// {attribute 'hide_all_locals'}
FUNCTION_BLOCK FB_Huawei_SmartLogger
VAR_INPUT PERSISTENT
	bEnable						: BOOL;				//True = Function is enabled, FALSE = Function is dissabled, no new Data
	sIPAdress					: STRING(15);		//IP Adress from the Inverter
	sint_ID_Iverter1			:SINT;				// ID of inveter 1
	sint_ID_Iverter2			:SINT;				// ID of inveter 2
	sint_ID_Iverter3			:SINT;				// ID of inveter 3
	sint_ID_Iverter4			:SINT;				// ID of inveter 4
	sint_ID_Iverter5			:SINT;				// ID of inveter 5
	sint_ID_Iverter6			:SINT;				// ID of inveter 6
	sint_ID_Iverter7			:SINT;				// ID of inveter 7
	sint_ID_Iverter8			:SINT;				// ID of inveter 8
	sint_ID_Iverter9			:SINT;				// ID of inveter 9
	sint_ID_Iverter10			:SINT;				// ID of inveter 10
	sint_ID_Iverter11			:SINT;				// ID of inveter 11
	sint_ID_Iverter12			:SINT;				// ID of inveter 12
	
	
END_VAR
VAR_OUTPUT
	st_Huawei_SmartLogger		: ARRAY[1..20] OF ST_Huawei_SmartLogger_OutData;					//Output structure with Data 
	stDataEMPower_PV			: ARRAY[1..20] OF ST_ElectricMeter_Output_Power;					//Output structure with Data from Electric Meter PV (Power Data)
	stDataEMCounter_PV 			: ARRAY[1..20] OF ST_ElectricMeter_Output_Counter;					//Output structure with Data from Electric Meter PV (Counter Data)
	diNrOfEM_OUT_PV				: DINT;																//Active Number from the Electric Meter for using on other functions
END_VAR
VAR
	sint_ID_Iverter				:ARRAY[1..12] OF SINT;				// Array of ID of inveter 
	fbMeter						: ARRAY[1..30] OF FB_ElectricMeter;					//Electric Meter Function 
	fbElMeter					: FB_ElectricMeter;									//Electric Meter Function for sumation values 
	
	fbNumberDevice				: FB_NumberOfDevice;								//Function block to calcualte the number of the Device
	fbConvertEnergyRegister		: FB_CV_WORD_TO_DWORD;								//Convert function
	fbMBRead_FC3				: FB_MBReadRegs;									//Modbus Read Function (FC3)
	timDelay					: TON;												//Timer for Delay between Requests
	timTimeout					: TON;												//Timer for Timeout
	timDissableFunctions		: TON;												//Timer to dissable the Function after Lynus_Standards.Constants_General.tTimeDissableLynusFunctions Days without connection to the Lynus Cloud
	timResetConnectionOnGVL		: TON;												//Timer to try reset the connection Flag on the GVL. (When somebody delete the Connection Function and make only a onlinechange)
	FPEnable					: R_TRIG;											//Internal positive Edge
	FPError_FC_3				: R_TRIG;											//Internal positive Edge
	PD_String					: FB_PersistentData_String;							//Function to save persistent data 
	stFloat						: ST_UN_FLOAT_CONVERT_DWORD_REAL;					//Convert the Float Raw Value
	arrBuffer_FC3				: ARRAY[0..25] OF WORD;							//Buffer with Data from FC3
	arrPD						: ARRAY[1..2] OF FB_PersistentData_Number;			//Function to save persistent data 
	byWaitInStep				: BYTE;												//Wait in Step before start to clean data on PLC
	iStateGVLData				: INT;												//State machine to handle the data on the GVL
	iStateModbus				: INT;												//State variable for Statemachine
	iStateModbus_CP				: INT;												//Compare State variable
	diCounterForGVL				: DINT;												//Counter to clean old data on GVL
	lrCheckValue				: LREAL;											//Internal Value to check the value before convert
	x							: INT;
	i: INT;
	int_Poll_Counter			: INT;												//Poll1 = inverter_ID 1,....
	byLPForInverter: INT;
	lrCounterEnergyProduction: LREAL;
	dwInput: DWORD;
	int_maxPolls				:INT :=12;											//maximum number of polls / inverter. 
	ton_Wait: Ton;
	FB_ConvertData			:FB_Convert_Huawei_SmartLogger;
	lreal1: LREAL;
	lreal2: LREAL;
	lreal3: LREAL;
	lreal4: LREAL;
	lreal5: LREAL;
	lreal6: LREAL;
	lreal7: LREAL;
	lreal8: LREAL;
	lreal9: LREAL;
	lreal10: LREAL;
	lreal11: LREAL;
	lreal12: LREAL;
	lreal13: LREAL;
	lreal14: LREAL;
	lreal15: LREAL;
	lreal16: LREAL;
	lreal17: LREAL;
	lreal18: LREAL;
	lreal19: LREAL;
	lreal20: LREAL;
	END_VAR

//Creator : Stefan Lackner
//Company : EfficientIO
//Date : 17.10.2022
//Version : 0.0.0.1		

//With this function its possible to read out values from the SmartLogger from the manufacturer Huawei
//This Function read out the Values from up to 12 inverters behind a SmartLogger. The SmartLogger could handle up to 247 inverters. 
//The protocol to the Inverter is Modbus TCP
//Attention. To access the registers, an offset of 1 must always be subtracted. Register 40001 would then be on register 40000.
//The document "SmartLogger ModBus Interface Definitions.pdf" issue 35 got used for the Modbus adress List

//NOTE for diNr.....Designation => 
//_IN = Here Data come in from other Functions or go out to other functions about the GVL
//_OUT = Here Data go out to other functions about the GVL


(*------------------------------------------------------------------------------------------General Input Part---------------------------------------------------------------------------------------------*)

//Check limitation
sint_ID_Iverter1 := LIMIT(0,sint_ID_Iverter1,127);
sint_ID_Iverter2 := LIMIT(0,sint_ID_Iverter2,127);
sint_ID_Iverter3 := LIMIT(0,sint_ID_Iverter3,127);
sint_ID_Iverter4 := LIMIT(0,sint_ID_Iverter4,127);
sint_ID_Iverter5 := LIMIT(0,sint_ID_Iverter5,127);
sint_ID_Iverter6 := LIMIT(0,sint_ID_Iverter6,127);
sint_ID_Iverter7 := LIMIT(0,sint_ID_Iverter7,127);
sint_ID_Iverter8 := LIMIT(0,sint_ID_Iverter8,127);
sint_ID_Iverter9 := LIMIT(0,sint_ID_Iverter9,127);
sint_ID_Iverter10:= LIMIT(0,sint_ID_Iverter10,127);
sint_ID_Iverter11:= LIMIT(0,sint_ID_Iverter11,127);
sint_ID_Iverter12 := LIMIT(0,sint_ID_Iverter12,127);
// copy in an array, easier for handling in the state maschine
sint_ID_Iverter[1]	:=	sint_ID_Iverter1;
sint_ID_Iverter[2]	:=	sint_ID_Iverter2;
sint_ID_Iverter[3]	:=	sint_ID_Iverter3;
sint_ID_Iverter[4]	:=	sint_ID_Iverter4;
sint_ID_Iverter[5]	:=	sint_ID_Iverter5;
sint_ID_Iverter[6]	:=	sint_ID_Iverter6;
sint_ID_Iverter[7]	:=	sint_ID_Iverter7;
sint_ID_Iverter[8]	:=	sint_ID_Iverter8;
sint_ID_Iverter[9]	:=	sint_ID_Iverter9;
sint_ID_Iverter[10]	:=	sint_ID_Iverter10;
sint_ID_Iverter[11]	:=	sint_ID_Iverter11;
sint_ID_Iverter[12]	:=	sint_ID_Iverter12;



(*-------------------------------------------------------------Calcualte the number of EM System---------------------------------------------------------------*)

fbNumberDevice(
	diActualNumberOfDevices:= Lynus_Standards.GVL_Energy.stNumberOfDevices.diNumberOfElectricMeters, 
	diMaxNumberOfDevices:= Constants_Energy.diMaxNumberOfElectricMeters, 
	udiCounterOnlineChange:= TwinCAT_SystemInfoVarList._AppInfo.OnlineChangeCnt, 
	bNumberIsCalculatet=> , 
	bFPNumberIsCalculatet=> , 
	bOnlineChange=> , 
	diNumberForThisDevice=> diNrOfEM_OUT_PV, 
	diNumberOfTotalDevices=> );

//Write new Numer on GVL
IF fbNumberDevice.bFPNumberIsCalculatet THEN
	Lynus_Standards.GVL_Energy.stNumberOfDevices.diNumberOfElectricMeters := fbNumberDevice.diNumberOfTotalDevices;	
END_IF 

//Delete old Number on GVL
IF fbNumberDevice.bOnlineChange THEN 
	Lynus_Standards.GVL_Energy.stNumberOfDevices.diNumberOfElectricMeters := diNrOfEM_OUT_PV;	
		iStateGVLData := 1; 
END_IF

(*-------------------------------------------------------------Service from Backend is ready and check the connection to backend for dissabel/enable Function---------------------------------------------------------------*)

//Try to reset the variable for connection on the GVL. When all is normal then the EfficientIO Mqtt connection function set this variable to true in the next cycle
//When we have no connection to the backend then after Lynus_Standards.Constants_General.tTimeDissableLynusFunctions days the Function is dissabled with all of his functionalities
timResetConnectionOnGVL(IN:= NOT timResetConnectionOnGVL.Q, PT:= T#1H, Q=> , ET=> );
IF timResetConnectionOnGVL.Q THEN 
	Lynus_Standards.GVL_Communicator.bStateConnectionToEnableFunctions := FALSE; 
END_IF
IF NOT Lynus_Standards.GVL_Communicator.bStateConnectionToEnableFunctions THEN 
	timDissableFunctions.IN := TRUE; 
ELSE 
	timDissableFunctions.IN := FALSE; 
END_IF  
timDissableFunctions(IN:= , PT:= Lynus_Standards.Constants_General.tTimeDissableLynusFunctions, Q=> , ET=> );
	
(*------------------------------------------------------------------------------------------State Machine---------------------------------------------------------------------------------------------*)
	
//Enable
FPEnable(CLK:= bEnable, Q=> );
IF FPEnable.Q AND iStateModbus = 0 THEN 
	iStateModbus := 1; 
END_IF
IF NOT bEnable OR timDissableFunctions.Q THEN 
	iStateModbus := 0; 
END_IF

//Timer for delay
timDelay(IN:= , PT:= T#100MS, Q=> , ET=> );	

//Timer for Timeout in Statemachine
IF iStateModbus = iStateModbus_CP THEN 
	timTimeout.IN := TRUE; 
ELSE 
	timTimeout.IN := FALSE; 
END_IF
IF iStateModbus = 0 THEN 
	timTimeout.IN := FALSE; 
END_IF
timTimeout(IN:= , PT:= T#20S, Q=> , ET=> );	


//Statemachine
CASE iStateModbus OF
	
	0://Init Step
		iStateModbus_CP := iStateModbus;
		timDelay.IN := FALSE;
		FOR i:=1 TO 20 BY 1 DO
			st_Huawei_SmartLogger[i].bFunctionIsActive := FALSE;
			st_Huawei_SmartLogger[i].eOperatingStateInverter := E_Huawei_SmartLogger_OperatingState.Unknown ;
		END_FOR
		
		fbMBRead_FC3.bExecute := FALSE;
		lrCheckValue := 0;
									
	1://Read out first inverter
		int_Poll_Counter:=1;			//Poll int_Poll_Counter : Inverter int_Poll_Counter 	
		st_Huawei_SmartLogger[int_Poll_Counter].bFunctionIsActive := TRUE;
		iStateModbus_CP := iStateModbus;
		fbMBRead_FC3.nQuantity := 25;
		fbMBRead_FC3.nMBAddr := (51000+(25*(SINT_TO_WORD(sint_ID_Iverter[int_Poll_Counter]) - 1)));
		fbMBRead_FC3.bExecute := TRUE;
			
		IF fbMBRead_FC3.bBusy THEN 
			timDelay.IN := TRUE; 
		END_IF
		
		//Wait for Delay, copy Data and then next step
		IF NOT fbMBRead_FC3.bBusy AND NOT fbMBRead_FC3.bError AND timDelay.Q THEN
			// convert received data
			FB_ConvertData(	arrBuffer_FC3			:=	arrBuffer_FC3,
											int_Poll_Counter		:=	int_Poll_Counter,
											lrPowerTotal			=>	fbMeter[int_Poll_Counter].lrPowerTotal,	
											lrReactivePowerTotal	=> 	fbMeter[int_Poll_Counter].lrReactivePowerTotal,
											eOperatingStateInverter	=>	st_Huawei_SmartLogger[int_Poll_Counter].eOperatingStateInverter);
	
			//Next Step
			fbMBRead_FC3.bExecute := FALSE;
			timDelay.IN := FALSE;
			iStateModbus := iStateModbus+1;
			IF arrBuffer_FC3[9]<>0 THEN
				st_Huawei_SmartLogger[int_Poll_Counter].bError := FALSE; 
				st_Huawei_SmartLogger[int_Poll_Counter].eErrorState := E_Huawei_SmartLogger_Error.eNoError;
			ELSE
				st_Huawei_SmartLogger[int_Poll_Counter].bError := FALSE; 
				st_Huawei_SmartLogger[int_Poll_Counter].eErrorState := E_Huawei_SmartLogger_Error.eNoError;
			END_IF
		END_IF
			
		//Error from Inverter 
		IF NOT fbMBRead_FC3.bBusy AND NOT fbMBRead_FC3.bError AND timDelay.Q AND arrBuffer_FC3[9] >= 16#0300 AND arrBuffer_FC3[9] <= 16#0308 THEN
			iStateModbus := 300;
			st_Huawei_SmartLogger[int_Poll_Counter].eErrorState := E_Huawei_SmartLogger_Error.eHuawei_SmartLoggerError;
		END_IF
	
		//Error or Timeout
		IF FPError_FC_3.Q OR timTimeout.Q THEN
			iStateModbus := 300;
			st_Huawei_SmartLogger[int_Poll_Counter].eOperatingStateInverter := E_Huawei_SmartLogger_OperatingState.Unknown;
			st_Huawei_SmartLogger[int_Poll_Counter].eErrorState	:=	E_Huawei_SmartLogger_Error.eModbusTCPError;
		END_IF
		
	2://Wait and go to step 1 or step 3
		iStateModbus_CP := iStateModbus;
		IF sint_ID_Iverter[int_Poll_Counter+1] = 0 OR int_Poll_Counter=int_maxPolls THEN		// if ID is not in use, go to state 100
			iStateModbus := 100;
		ELSE
			iStateModbus := 3;
			int_Poll_Counter:=int_Poll_Counter+1;			//Poll int_Poll_Counter : Inverter int_Poll_Counter 	
		END_IF

	3://Read out next inverter
		st_Huawei_SmartLogger[int_Poll_Counter].bFunctionIsActive := TRUE;
		iStateModbus_CP := iStateModbus;
		fbMBRead_FC3.nQuantity := 25;
		fbMBRead_FC3.nMBAddr := (51000+(25*(SINT_TO_WORD(sint_ID_Iverter[int_Poll_Counter]) - 1)));
		fbMBRead_FC3.bExecute := TRUE;
			
		IF fbMBRead_FC3.bBusy THEN 
			timDelay.IN := TRUE; 
		END_IF
		
		//Wait for Delay, copy Data and then next step
		IF NOT fbMBRead_FC3.bBusy AND NOT fbMBRead_FC3.bError AND timDelay.Q THEN
			// convert received data
			FB_ConvertData(	arrBuffer_FC3			:=	arrBuffer_FC3,
											int_Poll_Counter		:=	int_Poll_Counter,
											lrPowerTotal			=>	fbMeter[int_Poll_Counter].lrPowerTotal,	
											lrReactivePowerTotal	=> 	fbMeter[int_Poll_Counter].lrReactivePowerTotal,
											eOperatingStateInverter	=>	st_Huawei_SmartLogger[int_Poll_Counter].eOperatingStateInverter);
	
			//Next Step
			fbMBRead_FC3.bExecute := FALSE;
			timDelay.IN := FALSE;
			iStateModbus := iStateModbus+1;
			IF arrBuffer_FC3[9]<>0 THEN
				st_Huawei_SmartLogger[int_Poll_Counter].bError := FALSE; 
				st_Huawei_SmartLogger[int_Poll_Counter].eErrorState := E_Huawei_SmartLogger_Error.eNoError;
			ELSE
				st_Huawei_SmartLogger[int_Poll_Counter].bError := FALSE; 
				st_Huawei_SmartLogger[int_Poll_Counter].eErrorState := E_Huawei_SmartLogger_Error.eNoError;
			END_IF
		END_IF
			
		//Error from Inverter 
		IF NOT fbMBRead_FC3.bBusy AND NOT fbMBRead_FC3.bError AND timDelay.Q AND arrBuffer_FC3[9] >= 16#0300 AND arrBuffer_FC3[9] <= 16#0308 THEN
			iStateModbus := 300;
			st_Huawei_SmartLogger[int_Poll_Counter].eErrorState := E_Huawei_SmartLogger_Error.eHuawei_SmartLoggerError;
		END_IF
	
		//Error or Timeout
		IF FPError_FC_3.Q OR timTimeout.Q THEN
			iStateModbus := 300;
			st_Huawei_SmartLogger[int_Poll_Counter].eOperatingStateInverter := E_Huawei_SmartLogger_OperatingState.Unknown;
			st_Huawei_SmartLogger[int_Poll_Counter].eErrorState	:=	E_Huawei_SmartLogger_Error.eModbusTCPError;
		END_IF
		
	4://Wait and go to step +1 or step 100
		iStateModbus_CP := iStateModbus;
		IF sint_ID_Iverter[int_Poll_Counter+1] = 0 OR int_Poll_Counter=int_maxPolls THEN		// if ID is not in use, go to state 100
			iStateModbus := 100;
		ELSE
			iStateModbus := iStateModbus+1;
			int_Poll_Counter:=int_Poll_Counter+1;			//Poll int_Poll_Counter : Inverter int_Poll_Counter 	
		END_IF
	
	5://Read out next inverter
		st_Huawei_SmartLogger[int_Poll_Counter].bFunctionIsActive := TRUE;
		iStateModbus_CP := iStateModbus;
		fbMBRead_FC3.nQuantity := 25;
		fbMBRead_FC3.nMBAddr := (51000+(25*(SINT_TO_WORD(sint_ID_Iverter[int_Poll_Counter]) - 1)));
		fbMBRead_FC3.bExecute := TRUE;
			
		IF fbMBRead_FC3.bBusy THEN 
			timDelay.IN := TRUE; 
		END_IF
		
		//Wait for Delay, copy Data and then next step
		IF NOT fbMBRead_FC3.bBusy AND NOT fbMBRead_FC3.bError AND timDelay.Q THEN
			// convert received data
			FB_ConvertData(	arrBuffer_FC3			:=	arrBuffer_FC3,
											int_Poll_Counter		:=	int_Poll_Counter,
											lrPowerTotal			=>	fbMeter[int_Poll_Counter].lrPowerTotal,	
											lrReactivePowerTotal	=> 	fbMeter[int_Poll_Counter].lrReactivePowerTotal,
											eOperatingStateInverter	=>	st_Huawei_SmartLogger[int_Poll_Counter].eOperatingStateInverter);
	
			//Next Step
			fbMBRead_FC3.bExecute := FALSE;
			timDelay.IN := FALSE;
			iStateModbus := iStateModbus+1;
			IF arrBuffer_FC3[9]<>0 THEN
				st_Huawei_SmartLogger[int_Poll_Counter].bError := FALSE; 
				st_Huawei_SmartLogger[int_Poll_Counter].eErrorState := E_Huawei_SmartLogger_Error.eNoError;
			ELSE
				st_Huawei_SmartLogger[int_Poll_Counter].bError := FALSE; 
				st_Huawei_SmartLogger[int_Poll_Counter].eErrorState := E_Huawei_SmartLogger_Error.eNoError;
			END_IF
		END_IF
			
		//Error from Inverter 
		IF NOT fbMBRead_FC3.bBusy AND NOT fbMBRead_FC3.bError AND timDelay.Q AND arrBuffer_FC3[9] >= 16#0300 AND arrBuffer_FC3[9] <= 16#0308 THEN
			iStateModbus := 300;
			st_Huawei_SmartLogger[int_Poll_Counter].eErrorState := E_Huawei_SmartLogger_Error.eHuawei_SmartLoggerError;
		END_IF
	
		//Error or Timeout
		IF FPError_FC_3.Q OR timTimeout.Q THEN
			iStateModbus := 300;
			st_Huawei_SmartLogger[int_Poll_Counter].eOperatingStateInverter := E_Huawei_SmartLogger_OperatingState.Unknown;
			st_Huawei_SmartLogger[int_Poll_Counter].eErrorState	:=	E_Huawei_SmartLogger_Error.eModbusTCPError;
		END_IF
		
	6://Wait and go to step +1 or step 100
		iStateModbus_CP := iStateModbus;
		IF sint_ID_Iverter[int_Poll_Counter+1] = 0 OR int_Poll_Counter=int_maxPolls THEN		// if ID is not in use, go to state 100
			iStateModbus := 100;
		ELSE
			iStateModbus := iStateModbus+1;
			int_Poll_Counter:=int_Poll_Counter+1;			//Poll int_Poll_Counter : Inverter int_Poll_Counter 	
		END_IF
		
	7://Read out next inverter
		st_Huawei_SmartLogger[int_Poll_Counter].bFunctionIsActive := TRUE;
		iStateModbus_CP := iStateModbus;
		fbMBRead_FC3.nQuantity := 25;
		fbMBRead_FC3.nMBAddr := (51000+(25*(SINT_TO_WORD(sint_ID_Iverter[int_Poll_Counter]) - 1)));
		fbMBRead_FC3.bExecute := TRUE;
			
		IF fbMBRead_FC3.bBusy THEN 
			timDelay.IN := TRUE; 
		END_IF
		
		//Wait for Delay, copy Data and then next step
		IF NOT fbMBRead_FC3.bBusy AND NOT fbMBRead_FC3.bError AND timDelay.Q THEN
			// convert received data
			FB_ConvertData(	arrBuffer_FC3			:=	arrBuffer_FC3,
											int_Poll_Counter		:=	int_Poll_Counter,
											lrPowerTotal			=>	fbMeter[int_Poll_Counter].lrPowerTotal,	
											lrReactivePowerTotal	=> 	fbMeter[int_Poll_Counter].lrReactivePowerTotal,
											eOperatingStateInverter	=>	st_Huawei_SmartLogger[int_Poll_Counter].eOperatingStateInverter);
	
			//Next Step
			fbMBRead_FC3.bExecute := FALSE;
			timDelay.IN := FALSE;
			iStateModbus := iStateModbus+1;
			IF arrBuffer_FC3[9]<>0 THEN
				st_Huawei_SmartLogger[int_Poll_Counter].bError := FALSE; 
				st_Huawei_SmartLogger[int_Poll_Counter].eErrorState := E_Huawei_SmartLogger_Error.eNoError;
			ELSE
				st_Huawei_SmartLogger[int_Poll_Counter].bError := FALSE; 
				st_Huawei_SmartLogger[int_Poll_Counter].eErrorState := E_Huawei_SmartLogger_Error.eNoError;
			END_IF
		END_IF
			
		//Error from Inverter 
		IF NOT fbMBRead_FC3.bBusy AND NOT fbMBRead_FC3.bError AND timDelay.Q AND arrBuffer_FC3[9] >= 16#0300 AND arrBuffer_FC3[9] <= 16#0308 THEN
			iStateModbus := 300;
			st_Huawei_SmartLogger[int_Poll_Counter].eErrorState := E_Huawei_SmartLogger_Error.eHuawei_SmartLoggerError;
		END_IF
	
		//Error or Timeout
		IF FPError_FC_3.Q OR timTimeout.Q THEN
			iStateModbus := 300;
			st_Huawei_SmartLogger[int_Poll_Counter].eOperatingStateInverter := E_Huawei_SmartLogger_OperatingState.Unknown;
			st_Huawei_SmartLogger[int_Poll_Counter].eErrorState	:=	E_Huawei_SmartLogger_Error.eModbusTCPError;
		END_IF

	8://Wait and go to step +1 or step 100
		iStateModbus_CP := iStateModbus;
		IF sint_ID_Iverter[int_Poll_Counter+1] = 0 OR int_Poll_Counter=int_maxPolls THEN		// if ID is not in use, go to state 100
			iStateModbus := 100;
		ELSE
			iStateModbus := iStateModbus+1;
			int_Poll_Counter:=int_Poll_Counter+1;			//Poll int_Poll_Counter : Inverter int_Poll_Counter 	
		END_IF
		
	9://Read out next inverter
		st_Huawei_SmartLogger[int_Poll_Counter].bFunctionIsActive := TRUE;
		iStateModbus_CP := iStateModbus;
		fbMBRead_FC3.nQuantity := 25;
		fbMBRead_FC3.nMBAddr := (51000+(25*(SINT_TO_WORD(sint_ID_Iverter[int_Poll_Counter]) - 1)));
		fbMBRead_FC3.bExecute := TRUE;
			
		IF fbMBRead_FC3.bBusy THEN 
			timDelay.IN := TRUE; 
		END_IF
		
		//Wait for Delay, copy Data and then next step
		IF NOT fbMBRead_FC3.bBusy AND NOT fbMBRead_FC3.bError AND timDelay.Q THEN
			// convert received data
			FB_ConvertData(	arrBuffer_FC3			:=	arrBuffer_FC3,
											int_Poll_Counter		:=	int_Poll_Counter,
											lrPowerTotal			=>	fbMeter[int_Poll_Counter].lrPowerTotal,	
											lrReactivePowerTotal	=> 	fbMeter[int_Poll_Counter].lrReactivePowerTotal,
											eOperatingStateInverter	=>	st_Huawei_SmartLogger[int_Poll_Counter].eOperatingStateInverter);
	
			//Next Step
			fbMBRead_FC3.bExecute := FALSE;
			timDelay.IN := FALSE;
			iStateModbus := iStateModbus+1;
			IF arrBuffer_FC3[9]<>0 THEN
				st_Huawei_SmartLogger[int_Poll_Counter].bError := FALSE; 
				st_Huawei_SmartLogger[int_Poll_Counter].eErrorState := E_Huawei_SmartLogger_Error.eNoError;
			ELSE
				st_Huawei_SmartLogger[int_Poll_Counter].bError := FALSE; 
				st_Huawei_SmartLogger[int_Poll_Counter].eErrorState := E_Huawei_SmartLogger_Error.eNoError;
			END_IF
		END_IF
			
		//Error from Inverter 
		IF NOT fbMBRead_FC3.bBusy AND NOT fbMBRead_FC3.bError AND timDelay.Q AND arrBuffer_FC3[9] >= 16#0300 AND arrBuffer_FC3[9] <= 16#0308 THEN
			iStateModbus := 300;
			st_Huawei_SmartLogger[int_Poll_Counter].eErrorState := E_Huawei_SmartLogger_Error.eHuawei_SmartLoggerError;
		END_IF
	
		//Error or Timeout
		IF FPError_FC_3.Q OR timTimeout.Q THEN
			iStateModbus := 300;
			st_Huawei_SmartLogger[int_Poll_Counter].eOperatingStateInverter := E_Huawei_SmartLogger_OperatingState.Unknown;
			st_Huawei_SmartLogger[int_Poll_Counter].eErrorState	:=	E_Huawei_SmartLogger_Error.eModbusTCPError;
		END_IF
		
	10://Wait and go to step +1 or step 100
		iStateModbus_CP := iStateModbus;
		IF sint_ID_Iverter[int_Poll_Counter+1] = 0 OR int_Poll_Counter=int_maxPolls THEN		// if ID is not in use, go to state 100
			iStateModbus := 100;
		ELSE
			iStateModbus := iStateModbus+1;
			int_Poll_Counter:=int_Poll_Counter+1;			//Poll int_Poll_Counter : Inverter int_Poll_Counter 	
		END_IF
		
	11://Read out next inverter
		st_Huawei_SmartLogger[int_Poll_Counter].bFunctionIsActive := TRUE;
		iStateModbus_CP := iStateModbus;
		fbMBRead_FC3.nQuantity := 25;
		fbMBRead_FC3.nMBAddr := (51000+(25*(SINT_TO_WORD(sint_ID_Iverter[int_Poll_Counter]) - 1)));
		fbMBRead_FC3.bExecute := TRUE;
			
		IF fbMBRead_FC3.bBusy THEN 
			timDelay.IN := TRUE; 
		END_IF
		
		//Wait for Delay, copy Data and then next step
		IF NOT fbMBRead_FC3.bBusy AND NOT fbMBRead_FC3.bError AND timDelay.Q THEN
			// convert received data
			FB_ConvertData(	arrBuffer_FC3			:=	arrBuffer_FC3,
											int_Poll_Counter		:=	int_Poll_Counter,
											lrPowerTotal			=>	fbMeter[int_Poll_Counter].lrPowerTotal,	
											lrReactivePowerTotal	=> 	fbMeter[int_Poll_Counter].lrReactivePowerTotal,
											eOperatingStateInverter	=>	st_Huawei_SmartLogger[int_Poll_Counter].eOperatingStateInverter);
	
			//Next Step
			fbMBRead_FC3.bExecute := FALSE;
			timDelay.IN := FALSE;
			iStateModbus := iStateModbus+1;
			IF arrBuffer_FC3[9]<>0 THEN
				st_Huawei_SmartLogger[int_Poll_Counter].bError := FALSE; 
				st_Huawei_SmartLogger[int_Poll_Counter].eErrorState := E_Huawei_SmartLogger_Error.eNoError;
			ELSE
				st_Huawei_SmartLogger[int_Poll_Counter].bError := FALSE; 
				st_Huawei_SmartLogger[int_Poll_Counter].eErrorState := E_Huawei_SmartLogger_Error.eNoError;
			END_IF
		END_IF
			
		//Error from Inverter 
		IF NOT fbMBRead_FC3.bBusy AND NOT fbMBRead_FC3.bError AND timDelay.Q AND arrBuffer_FC3[9] >= 16#0300 AND arrBuffer_FC3[9] <= 16#0308 THEN
			iStateModbus := 300;
			st_Huawei_SmartLogger[int_Poll_Counter].eErrorState := E_Huawei_SmartLogger_Error.eHuawei_SmartLoggerError;
		END_IF
	
		//Error or Timeout
		IF FPError_FC_3.Q OR timTimeout.Q THEN
			iStateModbus := 300;
			st_Huawei_SmartLogger[int_Poll_Counter].eOperatingStateInverter := E_Huawei_SmartLogger_OperatingState.Unknown;
			st_Huawei_SmartLogger[int_Poll_Counter].eErrorState	:=	E_Huawei_SmartLogger_Error.eModbusTCPError;
		END_IF
		
	12://Wait and go to step +1 or step 100
		iStateModbus_CP := iStateModbus;
		IF sint_ID_Iverter[int_Poll_Counter+1] = 0 OR int_Poll_Counter=int_maxPolls THEN		// if ID is not in use, go to state 100
			iStateModbus := 100;
		ELSE
			iStateModbus := iStateModbus+1;
			int_Poll_Counter:=int_Poll_Counter+1;			//Poll int_Poll_Counter : Inverter int_Poll_Counter 	
		END_IF
		
	13://Read out next inverter
		st_Huawei_SmartLogger[int_Poll_Counter].bFunctionIsActive := TRUE;
		iStateModbus_CP := iStateModbus;
		fbMBRead_FC3.nQuantity := 25;
		fbMBRead_FC3.nMBAddr := (51000+(25*(SINT_TO_WORD(sint_ID_Iverter[int_Poll_Counter]) - 1)));
		fbMBRead_FC3.bExecute := TRUE;
			
		IF fbMBRead_FC3.bBusy THEN 
			timDelay.IN := TRUE; 
		END_IF
		
		//Wait for Delay, copy Data and then next step
		IF NOT fbMBRead_FC3.bBusy AND NOT fbMBRead_FC3.bError AND timDelay.Q THEN
			// convert received data
			FB_ConvertData(	arrBuffer_FC3			:=	arrBuffer_FC3,
											int_Poll_Counter		:=	int_Poll_Counter,
											lrPowerTotal			=>	fbMeter[int_Poll_Counter].lrPowerTotal,	
											lrReactivePowerTotal	=> 	fbMeter[int_Poll_Counter].lrReactivePowerTotal,
											eOperatingStateInverter	=>	st_Huawei_SmartLogger[int_Poll_Counter].eOperatingStateInverter);
	
			//Next Step
			fbMBRead_FC3.bExecute := FALSE;
			timDelay.IN := FALSE;
			iStateModbus := iStateModbus+1;
			IF arrBuffer_FC3[9]<>0 THEN
				st_Huawei_SmartLogger[int_Poll_Counter].bError := FALSE; 
				st_Huawei_SmartLogger[int_Poll_Counter].eErrorState := E_Huawei_SmartLogger_Error.eNoError;
			ELSE
				st_Huawei_SmartLogger[int_Poll_Counter].bError := FALSE; 
				st_Huawei_SmartLogger[int_Poll_Counter].eErrorState := E_Huawei_SmartLogger_Error.eNoError;
			END_IF
		END_IF
			
		//Error from Inverter 1
		IF NOT fbMBRead_FC3.bBusy AND NOT fbMBRead_FC3.bError AND timDelay.Q AND arrBuffer_FC3[9] >= 16#0300 AND arrBuffer_FC3[9] <= 16#0308 THEN
			iStateModbus := 300;
			st_Huawei_SmartLogger[int_Poll_Counter].eErrorState := E_Huawei_SmartLogger_Error.eHuawei_SmartLoggerError;
		END_IF
	
		//Error or Timeout
		IF FPError_FC_3.Q OR timTimeout.Q THEN
			iStateModbus := 300;
			st_Huawei_SmartLogger[int_Poll_Counter].eOperatingStateInverter := E_Huawei_SmartLogger_OperatingState.Unknown;
			st_Huawei_SmartLogger[int_Poll_Counter].eErrorState	:=	E_Huawei_SmartLogger_Error.eModbusTCPError;
		END_IF
		
	14://Wait and go to step +1 or step 100
		iStateModbus_CP := iStateModbus;
		IF sint_ID_Iverter[int_Poll_Counter+1] = 0 OR int_Poll_Counter=int_maxPolls THEN		// if ID is not in use, go to state 100
			iStateModbus := 100;
		ELSE
			iStateModbus := iStateModbus+1;
			int_Poll_Counter:=int_Poll_Counter+1;			//Poll int_Poll_Counter : Inverter int_Poll_Counter 	
		END_IF
		
	15://Read out next inverter
		st_Huawei_SmartLogger[int_Poll_Counter].bFunctionIsActive := TRUE;
		iStateModbus_CP := iStateModbus;
		fbMBRead_FC3.nQuantity := 25;
		fbMBRead_FC3.nMBAddr := (51000+(25*(SINT_TO_WORD(sint_ID_Iverter[int_Poll_Counter]) - 1)));
		fbMBRead_FC3.bExecute := TRUE;
			
		IF fbMBRead_FC3.bBusy THEN 
			timDelay.IN := TRUE; 
		END_IF
		
		//Wait for Delay, copy Data and then next step
		IF NOT fbMBRead_FC3.bBusy AND NOT fbMBRead_FC3.bError AND timDelay.Q THEN
			// convert received data
			FB_ConvertData(	arrBuffer_FC3			:=	arrBuffer_FC3,
											int_Poll_Counter		:=	int_Poll_Counter,
											lrPowerTotal			=>	fbMeter[int_Poll_Counter].lrPowerTotal,	
											lrReactivePowerTotal	=> 	fbMeter[int_Poll_Counter].lrReactivePowerTotal,
											eOperatingStateInverter	=>	st_Huawei_SmartLogger[int_Poll_Counter].eOperatingStateInverter);
	
			//Next Step
			fbMBRead_FC3.bExecute := FALSE;
			timDelay.IN := FALSE;
			iStateModbus := iStateModbus+1;
			IF arrBuffer_FC3[9]<>0 THEN
				st_Huawei_SmartLogger[int_Poll_Counter].bError := FALSE; 
				st_Huawei_SmartLogger[int_Poll_Counter].eErrorState := E_Huawei_SmartLogger_Error.eNoError;
			ELSE
				st_Huawei_SmartLogger[int_Poll_Counter].bError := FALSE; 
				st_Huawei_SmartLogger[int_Poll_Counter].eErrorState := E_Huawei_SmartLogger_Error.eNoError;
			END_IF
		END_IF
			
		//Error from Inverter 
		IF NOT fbMBRead_FC3.bBusy AND NOT fbMBRead_FC3.bError AND timDelay.Q AND arrBuffer_FC3[9] >= 16#0300 AND arrBuffer_FC3[9] <= 16#0308 THEN
			iStateModbus := 300;
			st_Huawei_SmartLogger[int_Poll_Counter].eErrorState := E_Huawei_SmartLogger_Error.eHuawei_SmartLoggerError;
		END_IF
	
		//Error or Timeout
		IF FPError_FC_3.Q OR timTimeout.Q THEN
			iStateModbus := 300;
			st_Huawei_SmartLogger[int_Poll_Counter].eOperatingStateInverter := E_Huawei_SmartLogger_OperatingState.Unknown;
			st_Huawei_SmartLogger[int_Poll_Counter].eErrorState	:=	E_Huawei_SmartLogger_Error.eModbusTCPError;
		END_IF
		
	16://Wait and go to step +1 or step 100
		iStateModbus_CP := iStateModbus;
		IF sint_ID_Iverter[int_Poll_Counter+1] = 0 OR int_Poll_Counter=int_maxPolls THEN		// if ID is not in use, go to state 100
			iStateModbus := 100;
		ELSE
			iStateModbus := iStateModbus+1;
			int_Poll_Counter:=int_Poll_Counter+1;			//Poll int_Poll_Counter : Inverter int_Poll_Counter 	
		END_IF

	17://Read out next inverter
		st_Huawei_SmartLogger[int_Poll_Counter].bFunctionIsActive := TRUE;
		iStateModbus_CP := iStateModbus;
		fbMBRead_FC3.nQuantity := 25;
		fbMBRead_FC3.nMBAddr := (51000+(25*(SINT_TO_WORD(sint_ID_Iverter[int_Poll_Counter]) - 1)));
		fbMBRead_FC3.bExecute := TRUE;
			
		IF fbMBRead_FC3.bBusy THEN 
			timDelay.IN := TRUE; 
		END_IF
		
		//Wait for Delay, copy Data and then next step
		IF NOT fbMBRead_FC3.bBusy AND NOT fbMBRead_FC3.bError AND timDelay.Q THEN
			// convert received data
			FB_ConvertData(	arrBuffer_FC3			:=	arrBuffer_FC3,
											int_Poll_Counter		:=	int_Poll_Counter,
											lrPowerTotal			=>	fbMeter[int_Poll_Counter].lrPowerTotal,	
											lrReactivePowerTotal	=> 	fbMeter[int_Poll_Counter].lrReactivePowerTotal,
											eOperatingStateInverter	=>	st_Huawei_SmartLogger[int_Poll_Counter].eOperatingStateInverter);
	
			//Next Step
			fbMBRead_FC3.bExecute := FALSE;
			timDelay.IN := FALSE;
			iStateModbus := iStateModbus+1;
			IF arrBuffer_FC3[9]<>0 THEN
				st_Huawei_SmartLogger[int_Poll_Counter].bError := FALSE; 
				st_Huawei_SmartLogger[int_Poll_Counter].eErrorState := E_Huawei_SmartLogger_Error.eNoError;
			ELSE
				st_Huawei_SmartLogger[int_Poll_Counter].bError := FALSE; 
				st_Huawei_SmartLogger[int_Poll_Counter].eErrorState := E_Huawei_SmartLogger_Error.eNoError;
			END_IF
		END_IF
			
		//Error from Inverter 
		IF NOT fbMBRead_FC3.bBusy AND NOT fbMBRead_FC3.bError AND timDelay.Q AND arrBuffer_FC3[9] >= 16#0300 AND arrBuffer_FC3[9] <= 16#0308 THEN
			iStateModbus := 300;
			st_Huawei_SmartLogger[int_Poll_Counter].eErrorState := E_Huawei_SmartLogger_Error.eHuawei_SmartLoggerError;
		END_IF
	
		//Error or Timeout
		IF FPError_FC_3.Q OR timTimeout.Q THEN
			iStateModbus := 300;
			st_Huawei_SmartLogger[int_Poll_Counter].eOperatingStateInverter := E_Huawei_SmartLogger_OperatingState.Unknown;
			st_Huawei_SmartLogger[int_Poll_Counter].eErrorState	:=	E_Huawei_SmartLogger_Error.eModbusTCPError;
		END_IF
		
	18://Wait and go to step +1 or step 100
		iStateModbus_CP := iStateModbus;
		IF sint_ID_Iverter[int_Poll_Counter+1] = 0 OR int_Poll_Counter=int_maxPolls THEN		// if ID is not in use, go to state 100
			iStateModbus := 100;
		ELSE
			iStateModbus := iStateModbus+1;
			int_Poll_Counter:=int_Poll_Counter+1;			//Poll int_Poll_Counter : Inverter int_Poll_Counter 	
		END_IF
		
	19://Read out next inverter
		st_Huawei_SmartLogger[int_Poll_Counter].bFunctionIsActive := TRUE;
		iStateModbus_CP := iStateModbus;
		fbMBRead_FC3.nQuantity := 25;
		fbMBRead_FC3.nMBAddr := (51000+(25*(SINT_TO_WORD(sint_ID_Iverter[int_Poll_Counter]) - 1)));
		fbMBRead_FC3.bExecute := TRUE;
			
		IF fbMBRead_FC3.bBusy THEN 
			timDelay.IN := TRUE; 
		END_IF
		
		//Wait for Delay, copy Data and then next step
		IF NOT fbMBRead_FC3.bBusy AND NOT fbMBRead_FC3.bError AND timDelay.Q THEN
			// convert received data
			FB_ConvertData(	arrBuffer_FC3			:=	arrBuffer_FC3,
											int_Poll_Counter		:=	int_Poll_Counter,
											lrPowerTotal			=>	fbMeter[int_Poll_Counter].lrPowerTotal,	
											lrReactivePowerTotal	=> 	fbMeter[int_Poll_Counter].lrReactivePowerTotal,
											eOperatingStateInverter	=>	st_Huawei_SmartLogger[int_Poll_Counter].eOperatingStateInverter);
	
			//Next Step
			fbMBRead_FC3.bExecute := FALSE;
			timDelay.IN := FALSE;
			iStateModbus := iStateModbus+1;
			IF arrBuffer_FC3[9]<>0 THEN
				st_Huawei_SmartLogger[int_Poll_Counter].bError := FALSE; 
				st_Huawei_SmartLogger[int_Poll_Counter].eErrorState := E_Huawei_SmartLogger_Error.eNoError;
			ELSE
				st_Huawei_SmartLogger[int_Poll_Counter].bError := FALSE; 
				st_Huawei_SmartLogger[int_Poll_Counter].eErrorState := E_Huawei_SmartLogger_Error.eNoError;
			END_IF
		END_IF
			
		//Error or Timeout
		IF FPError_FC_3.Q OR timTimeout.Q THEN
			iStateModbus := 300;
			st_Huawei_SmartLogger[int_Poll_Counter].eOperatingStateInverter := E_Huawei_SmartLogger_OperatingState.Unknown;
			st_Huawei_SmartLogger[int_Poll_Counter].eErrorState	:=	E_Huawei_SmartLogger_Error.eModbusTCPError;
		END_IF
	
		//Error or Timeout
		IF FPError_FC_3.Q OR timTimeout.Q THEN
			iStateModbus := 300;
			st_Huawei_SmartLogger[int_Poll_Counter].eOperatingStateInverter := E_Huawei_SmartLogger_Error.eModbusTCPError;
		END_IF

	20://Wait and go to step +1 or step 100
		iStateModbus_CP := iStateModbus;
		IF sint_ID_Iverter[int_Poll_Counter+1] = 0 OR int_Poll_Counter=int_maxPolls THEN		// if ID is not in use, go to state 100
			iStateModbus := 100;
		ELSE
			iStateModbus := iStateModbus+1;
			int_Poll_Counter:=int_Poll_Counter+1;			//Poll int_Poll_Counter : Inverter int_Poll_Counter 	
		END_IF

	21://Read out next inverter
		st_Huawei_SmartLogger[int_Poll_Counter].bFunctionIsActive := TRUE;
		iStateModbus_CP := iStateModbus;
		fbMBRead_FC3.nQuantity := 25;
		fbMBRead_FC3.nMBAddr := (51000+(25*(SINT_TO_WORD(sint_ID_Iverter[int_Poll_Counter]) - 1)));
		fbMBRead_FC3.bExecute := TRUE;
			
		IF fbMBRead_FC3.bBusy THEN 
			timDelay.IN := TRUE; 
		END_IF
		
		//Wait for Delay, copy Data and then next step
		IF NOT fbMBRead_FC3.bBusy AND NOT fbMBRead_FC3.bError AND timDelay.Q THEN
			// convert received data
			FB_ConvertData(	arrBuffer_FC3			:=	arrBuffer_FC3,
											int_Poll_Counter		:=	int_Poll_Counter,
											lrPowerTotal			=>	fbMeter[int_Poll_Counter].lrPowerTotal,	
											lrReactivePowerTotal	=> 	fbMeter[int_Poll_Counter].lrReactivePowerTotal,
											eOperatingStateInverter	=>	st_Huawei_SmartLogger[int_Poll_Counter].eOperatingStateInverter);
	
			//Next Step
			fbMBRead_FC3.bExecute := FALSE;
			timDelay.IN := FALSE;
			iStateModbus := iStateModbus+1;
			IF arrBuffer_FC3[9]<>0 THEN
				st_Huawei_SmartLogger[int_Poll_Counter].bError := FALSE; 
				st_Huawei_SmartLogger[int_Poll_Counter].eErrorState := E_Huawei_SmartLogger_Error.eNoError;
			ELSE
				st_Huawei_SmartLogger[int_Poll_Counter].bError := FALSE; 
				st_Huawei_SmartLogger[int_Poll_Counter].eErrorState := E_Huawei_SmartLogger_Error.eNoError;
			END_IF
		END_IF
			
		//Error from Inverter 
		IF NOT fbMBRead_FC3.bBusy AND NOT fbMBRead_FC3.bError AND timDelay.Q AND arrBuffer_FC3[9] >= 16#0300 AND arrBuffer_FC3[9] <= 16#0308 THEN
			iStateModbus := 300;
			st_Huawei_SmartLogger[int_Poll_Counter].eErrorState := E_Huawei_SmartLogger_Error.eHuawei_SmartLoggerError;
		END_IF
	
		//Error or Timeout
		IF FPError_FC_3.Q OR timTimeout.Q THEN
			iStateModbus := 300;
			st_Huawei_SmartLogger[int_Poll_Counter].eOperatingStateInverter := E_Huawei_SmartLogger_OperatingState.Unknown;
			st_Huawei_SmartLogger[int_Poll_Counter].eErrorState	:=	E_Huawei_SmartLogger_Error.eModbusTCPError;
		END_IF
		
	22://Wait and go to step +1 or step 100
		iStateModbus_CP := iStateModbus;
		IF sint_ID_Iverter[int_Poll_Counter+1] = 0 OR int_Poll_Counter=int_maxPolls THEN		// if ID is not in use, go to state 100
			iStateModbus := 100;
		ELSE
			iStateModbus := iStateModbus+1;
			int_Poll_Counter:=int_Poll_Counter+1;			//Poll int_Poll_Counter : Inverter int_Poll_Counter 	
		END_IF

	23://Read out next inverter
		st_Huawei_SmartLogger[int_Poll_Counter].bFunctionIsActive := TRUE;
		iStateModbus_CP := iStateModbus;
		fbMBRead_FC3.nQuantity := 25;
		fbMBRead_FC3.nMBAddr := (51000+(25*(SINT_TO_WORD(sint_ID_Iverter[int_Poll_Counter]) - 1)));
		fbMBRead_FC3.bExecute := TRUE;
			
		IF fbMBRead_FC3.bBusy THEN 
			timDelay.IN := TRUE; 
		END_IF
		
		//Wait for Delay, copy Data and then next step
		IF NOT fbMBRead_FC3.bBusy AND NOT fbMBRead_FC3.bError AND timDelay.Q THEN
			// convert received data
			FB_ConvertData(	arrBuffer_FC3			:=	arrBuffer_FC3,
											int_Poll_Counter		:=	int_Poll_Counter,
											lrPowerTotal			=>	fbMeter[int_Poll_Counter].lrPowerTotal,	
											lrReactivePowerTotal	=> 	fbMeter[int_Poll_Counter].lrReactivePowerTotal,
											eOperatingStateInverter	=>	st_Huawei_SmartLogger[int_Poll_Counter].eOperatingStateInverter);
	
			//Next Step
			fbMBRead_FC3.bExecute := FALSE;
			timDelay.IN := FALSE;
			iStateModbus := iStateModbus+1;
			IF arrBuffer_FC3[9]<>0 THEN
				st_Huawei_SmartLogger[int_Poll_Counter].bError := FALSE; 
				st_Huawei_SmartLogger[int_Poll_Counter].eErrorState := E_Huawei_SmartLogger_Error.eNoError;
			ELSE
				st_Huawei_SmartLogger[int_Poll_Counter].bError := FALSE; 
				st_Huawei_SmartLogger[int_Poll_Counter].eErrorState := E_Huawei_SmartLogger_Error.eNoError;
			END_IF
		END_IF
			
		//Error from Inverter 
		IF NOT fbMBRead_FC3.bBusy AND NOT fbMBRead_FC3.bError AND timDelay.Q AND arrBuffer_FC3[9] >= 16#0300 AND arrBuffer_FC3[9] <= 16#0308 THEN
			iStateModbus := 300;
			st_Huawei_SmartLogger[int_Poll_Counter].eErrorState := E_Huawei_SmartLogger_Error.eHuawei_SmartLoggerError;
		END_IF
	
		//Error or Timeout
		IF FPError_FC_3.Q OR timTimeout.Q THEN
			iStateModbus := 300;
			st_Huawei_SmartLogger[int_Poll_Counter].eOperatingStateInverter := E_Huawei_SmartLogger_OperatingState.Unknown;
			st_Huawei_SmartLogger[int_Poll_Counter].eErrorState	:=	E_Huawei_SmartLogger_Error.eModbusTCPError;
		END_IF
		
	24://Wait and go to step +1 or step 100
		iStateModbus_CP := iStateModbus;
		IF sint_ID_Iverter[int_Poll_Counter+1] = 0 OR int_Poll_Counter=int_maxPolls THEN		// if ID is not in use, go to state 100
			iStateModbus := 100;
		ELSE
			iStateModbus := iStateModbus+1;
			int_Poll_Counter:=int_Poll_Counter+1;			//Poll int_Poll_Counter : Inverter int_Poll_Counter 	
		END_IF




		
		
		
	100://Wait and go to step 1 
		iStateModbus_CP := iStateModbus;
		ton_Wait.In:=TRUE;
		IF ton_Wait.Q THEN
			ton_Wait.In:=FALSE;
			iStateModbus := 1;
		END_IF
			
	300://Error
		iStateModbus_CP := iStateModbus;
		timDelay.IN := FALSE;
		fbMBRead_FC3.bExecute := FALSE;
		st_Huawei_SmartLogger[int_Poll_Counter].bError := TRUE;
		ton_Wait.In:=TRUE;
		IF ton_Wait.Q THEN
			ton_Wait.In:=FALSE;
			iStateModbus := 1;
		END_IF
END_CASE

// wait timer
ton_Wait(PT:=T#2S);

	

(*------------------------------------------------------------------------------------------Modbus TCP Function---------------------------------------------------------------------------------------------*)

fbMBRead_FC3(	sIPAddr:= sIPAdress, 
				nTCPPort:= 502, 
				nUnitID := 0,
				cbLength:= SIZEOF(arrBuffer_FC3), 
				pDestAddr:= ADR(arrBuffer_FC3), 
				tTimeout:= T#10S );

FPError_FC_3(CLK:= fbMBRead_FC3.bError, Q=> );

(*----------------------------------------------------------------------------------------Electric Meter Data----------------------------------------------------------------------------------------------*)

//Error and Warning
FOR x:=1 TO 20 BY 1 DO
	IF timDissableFunctions.Q THEN 
		fbMeter[x].bWarning := TRUE; 
		fbMeter[x].iWarningCode := 0; 
	ELSE 
		fbMeter[x].bWarning := FALSE; 
	END_IF   

	IF st_Huawei_SmartLogger[x].bError OR Lynus_Standards.GVL_Energy.stNumberOfDevices.diNumberOfElectricMeters > Constants_Energy.diMaxNumberOfElectricMeters THEN 
		fbMeter[x].bError := TRUE; 
	ELSE 
		fbMeter[x].bError := FALSE; 
	END_IF  

	IF Lynus_Standards.GVL_Energy.stNumberOfDevices.diNumberOfElectricMeters > Constants_Energy.diMaxNumberOfElectricMeters THEN 
		fbMeter[x].iErrorCode := 1;
	ELSIF st_Huawei_SmartLogger[x].bError THEN 
		fbMeter[x].iErrorCode := 0;
	END_IF  

	//Function block for meter data
	fbMeter[x](
		bEnable:= bEnable AND NOT timDissableFunctions.Q, 
		bError:= , 
		bEnableReadOutFunction:= TRUE, 
		bWriteWithDelay:= TRUE,
		bPowerDataInvers:= TRUE, 
		bReadOutDataDone:= TRUE,
		iTimeReadOutInterval:= , 
		iErrorCode:= , 
		iWarningCode:= , 
		lrTotalCounterEnergy_Consumption:= 0, 
		lrTotalCounterEnergy_Production:= , 
		lrCounterEnergyT1_Consumption:= 0, 
		lrCounterEnergyT2_Consumption:= 0, 
		lrCounterEnergyT1_Production:= , 
		lrCounterEnergyT2_Production:= 0, 
		lrCurrentL1:= , 
		lrVoltageL1N:= , 
		lrVoltageL1L2:= , 
		lrPowerL1:= 0, 
		lrCurrentL2:= , 
		lrVoltageL2N:= , 
		lrVoltageL2L3:= , 
		lrPowerL2:= 0, 
		lrCurrentL3:= , 
		lrVoltageL3N:= , 
		lrVoltageL3L1:= , 
		lrPowerL3:= 0, 
		lrPowerTotal:= , 
		lrFrequency:= , 
		lrReactivePowerTotal:= , 
		lrApparentPowerTotal:= , 
		tTimDelayOutput:= T#5S, 
		stDataEMOutPower=> , 
		stDataEMOutPowerDelay=> stDataEMPower_PV[x], 
		stDataEMOutCounter=> ,
		stDataEMOutCounterDelay=> stDataEMCounter_PV[x], 
		bReadOutMeter=> );

END_FOR
//Read Out Data done for EM Function
IF NOT fbMBRead_FC3.bBusy AND NOT fbMBRead_FC3.bError THEN 
	fbMeter[int_Poll_Counter].bReadOutDataDone := TRUE;
ELSE 
	fbMeter[int_Poll_Counter].bReadOutDataDone := FALSE;
END_IF



(*-----------------------------------------------------------Handle data to Global structure for the Electric Meter system-----------------------------------------------------------------*)

CASE iStateGVLData OF
	
	0://Init Step
		byWaitInStep := 0;
		diCounterForGVL := 1;
	
	1://Wait for 4 Steps before clean al Data on GVL
		byWaitInStep := byWaitInStep + 1;
		IF byWaitInStep >= 4 AND fbNumberDevice.bNumberIsCalculatet THEN 
			iStateGVLData := 2; 
		END_IF
		//To much Devices, back to the Init step
		IF byWaitInStep >= 4 AND NOT fbNumberDevice.bNumberIsCalculatet THEN 
			iStateGVLData := 0; 
		END_IF	
			
	2://Clear all Data in GVL
		Lynus_Standards.GVL_Energy.stDataElectricMeters[diCounterForGVL].bEnabled := FALSE;	
		Lynus_Standards.GVL_Energy.stDataElectricMeters[diCounterForGVL].byErrorWarning := 0;
		Lynus_Standards.GVL_Energy.stDataElectricMeters[diCounterForGVL].lrCounterEnergyT1_Consumption := 0;
		Lynus_Standards.GVL_Energy.stDataElectricMeters[diCounterForGVL].lrCounterEnergyT1_Production := 0;
		Lynus_Standards.GVL_Energy.stDataElectricMeters[diCounterForGVL].lrCounterEnergyT2_Consumption := 0;
		Lynus_Standards.GVL_Energy.stDataElectricMeters[diCounterForGVL].lrCounterEnergyT2_Production := 0;
		Lynus_Standards.GVL_Energy.stDataElectricMeters[diCounterForGVL].lrPower := 0;
		Lynus_Standards.GVL_Energy.stDataElectricMeters[diCounterForGVL].lrPowerConsumption := 0;
		Lynus_Standards.GVL_Energy.stDataElectricMeters[diCounterForGVL].lrPowerConsumption := 0;
		Lynus_Standards.GVL_Energy.stDataElectricMeters[diCounterForGVL].lrPowerProduction := 0;
		Lynus_Standards.GVL_Energy.stDataElectricMeters[diCounterForGVL].lrTotalCounterEnergy_Consumption := 0;
		Lynus_Standards.GVL_Energy.stDataElectricMeters[diCounterForGVL].lrTotalCounterEnergy_Production := 0;
		
		diCounterForGVL := diCounterForGVL + 1;
		diCounterForGVL := LIMIT(0,diCounterForGVL,Constants_Energy.diMaxNumberOfElectricMeters);
		//Back to the init step
		IF diCounterForGVL >= Constants_Energy.diMaxNumberOfElectricMeters THEN 
			iStateGVLData := 0; 
		END_IF
END_CASE 	 

IF diNrOfEM_OUT_PV > 0 AND fbNumberDevice.bNumberIsCalculatet THEN
	Lynus_Standards.GVL_Energy.stDataElectricMeters[diNrOfEM_OUT_PV].bEnabled := fbElMeter.stDataEMOutPower.bEnabled;
	Lynus_Standards.GVL_Energy.stDataElectricMeters[diNrOfEM_OUT_PV].byErrorWarning := fbElMeter.stDataEMOutPower.byErrorWarning;
	Lynus_Standards.GVL_Energy.stDataElectricMeters[diNrOfEM_OUT_PV].lrCounterEnergyT1_Consumption := fbElMeter.stDataEMOutCounter.lrCounterEnergyT1_Consumption;
	Lynus_Standards.GVL_Energy.stDataElectricMeters[diNrOfEM_OUT_PV].lrCounterEnergyT1_Production := fbElMeter.stDataEMOutCounter.lrCounterEnergyT1_Production;
	Lynus_Standards.GVL_Energy.stDataElectricMeters[diNrOfEM_OUT_PV].lrCounterEnergyT2_Consumption := fbElMeter.stDataEMOutCounter.lrCounterEnergyT2_Consumption;
	Lynus_Standards.GVL_Energy.stDataElectricMeters[diNrOfEM_OUT_PV].lrCounterEnergyT2_Production := fbElMeter.stDataEMOutCounter.lrCounterEnergyT2_Production;		
	Lynus_Standards.GVL_Energy.stDataElectricMeters[diNrOfEM_OUT_PV].lrPower := fbElMeter.lrPowerTotal; // fbElMeter.stDataEMOutPower.lrPowerTotal;
	Lynus_Standards.GVL_Energy.stDataElectricMeters[diNrOfEM_OUT_PV].lrPowerConsumption := fbElMeter.stDataEMOutPower.lrPowerConsumption;
	Lynus_Standards.GVL_Energy.stDataElectricMeters[diNrOfEM_OUT_PV].lrPowerProduction := fbElMeter.stDataEMOutPower.lrPowerProduction;
	Lynus_Standards.GVL_Energy.stDataElectricMeters[diNrOfEM_OUT_PV].lrTotalCounterEnergy_Consumption := fbElMeter.stDataEMOutCounter.lrTotalCounterEnergy_Consumption;
	Lynus_Standards.GVL_Energy.stDataElectricMeters[diNrOfEM_OUT_PV].lrTotalCounterEnergy_Production := fbElMeter.stDataEMOutCounter.lrTotalCounterEnergy_Production;
END_IF


// Sum values for Meter
fbElMeter.lrPowerTotal := 0;
FOR byLPForInverter := 1 TO 20 BY 1 DO 
	lrCounterEnergyProduction := lrCounterEnergyProduction + fbMeter[byLPForInverter].stDataEMOutCounterDelay.lrTotalCounterEnergy_Production;
	IF lrCounterEnergyProduction > fbElMeter.lrCounterEnergyT1_Production THEN
		fbElMeter.lrCounterEnergyT1_Production := lrCounterEnergyProduction;
	END_IF
	fbElMeter.lrPowerTotal := fbElMeter.lrPowerTotal + fbMeter[byLPForInverter].stDataEMOutPowerDelay.lrPowerTotal;
END_FOR	
					
fbElMeter.lrTotalCounterEnergy_Production := fbElMeter.lrCounterEnergyT1_Production; 
fbElMeter(bEnable:=TRUE);


lreal1:=fbMeter[1].stDataEMOutPowerDelay.lrPowerTotal;
lreal2:=fbMeter[2].stDataEMOutPowerDelay.lrPowerTotal;
lreal3:=fbMeter[3].stDataEMOutPowerDelay.lrPowerTotal;
lreal4:=fbMeter[4].stDataEMOutPowerDelay.lrPowerTotal;
lreal5:=fbMeter[5].stDataEMOutPowerDelay.lrPowerTotal;
lreal6:=fbMeter[6].stDataEMOutPowerDelay.lrPowerTotal;
lreal7:=fbMeter[7].stDataEMOutPowerDelay.lrPowerTotal;
lreal8:=fbMeter[8].stDataEMOutPowerDelay.lrPowerTotal;
lreal9:=fbMeter[9].stDataEMOutPowerDelay.lrPowerTotal;
lreal10:=fbMeter[10].stDataEMOutPowerDelay.lrPowerTotal;
lreal11:=fbMeter[11].stDataEMOutPowerDelay.lrPowerTotal;
lreal12:=fbMeter[12].stDataEMOutPowerDelay.lrPowerTotal;
lreal13:=fbMeter[13].stDataEMOutPowerDelay.lrPowerTotal;
lreal14:=fbMeter[14].stDataEMOutPowerDelay.lrPowerTotal;
lreal15:=fbMeter[15].stDataEMOutPowerDelay.lrPowerTotal;
lreal16:=fbMeter[16].stDataEMOutPowerDelay.lrPowerTotal;
lreal17:=fbMeter[17].stDataEMOutPowerDelay.lrPowerTotal;
lreal18:=fbMeter[18].stDataEMOutPowerDelay.lrPowerTotal;
lreal19:=fbMeter[19].stDataEMOutPowerDelay.lrPowerTotal;
lreal20:=fbMeter[20].stDataEMOutPowerDelay.lrPowerTotal;

(*----------------------------------------------------------Save persistent data----------------------------------------------------------------*)

// arrPD[1](lrValue:= BOOL_TO_LREAL(bEnable), bEventBasedActive=> );
// arrPD[2](lrValue:= BYTE_TO_LREAL(byAmountOfInverters), bEventBasedActive=> );
PD_String(sText:= sIPAdress, bEventBasedActive=> );

END_FUNCTION_BLOCK

(* stored: Version 1.1.0.1, ProductVersion 3.1.4024.11
   POU FB_Huawei_SmartLogger: Id {b4c12ce6-c6bb-4362-a4da-542ebf2a554d}, SpecialFunc None *)
